INTERFACE PUBLIC MoveVelocityBuilder EXTENDS __System.IQueryInterface

METHOD PUBLIC Acceleration : MoveVelocityBuilder
VAR_INPUT
	value : LREAL;
END_VAR
END_METHOD

METHOD PUBLIC BufferMode : MoveVelocityBuilder
VAR_INPUT
	mode : MotionBufferMode;
END_VAR
END_METHOD

METHOD PUBLIC BuildMoveVelocityCommand : MotionCommand
VAR_INPUT
	axis : Axis;
END_VAR
END_METHOD

METHOD PUBLIC Deceleration : MoveVelocityBuilder
VAR_INPUT
	value : LREAL;
END_VAR
END_METHOD

METHOD PUBLIC Distance : MoveRelativeBuilder
VAR_INPUT
	value : LREAL;
END_VAR
END_METHOD

METHOD PUBLIC Jerk : MoveVelocityBuilder
VAR_INPUT
	value : LREAL;
END_VAR
END_METHOD

METHOD PUBLIC Position : MoveAbsoluteBuilder
VAR_INPUT
	value : LREAL;
END_VAR
END_METHOD

METHOD PUBLIC Velocity : MoveVelocityBuilder
VAR_INPUT
	value : LREAL;
END_VAR
END_METHOD

END_INTERFACE

(* stored: Version 1.1.0.1
   Itf MoveVelocityBuilder: Id {af81a36f-91e0-4229-8050-674aaf4d51c8}
   Folder Builders: Id {7fd778aa-403b-4bcf-b94b-ddb110cd0772}
   Folder PropertySetters: Id {c78165b8-d771-464a-881b-28b518193161}
   Method Acceleration: Id {1a50edb1-113b-4f46-83c6-b8f26a71a15e}
   Method BufferMode: Id {6a4f0400-b046-43df-b9ee-74e7ee22d50a}
   Method BuildMoveVelocityCommand: Id {0fd3c392-d1e2-06f3-2fa5-d8869d117ef5}
   Method Deceleration: Id {2885aa42-90e4-4613-82d7-1c22ebf0dd39}
   Method Distance: Id {492191b7-499f-40fe-a63e-283905023ebf}
   Method Jerk: Id {d31e94a9-727f-4bfb-bd51-0dd8ad61940f}
   Method Position: Id {2aad1022-9d1b-4af0-bc07-544790ecfdea}
   Method Velocity: Id {eb1b270e-f436-450a-b153-6c07dbc75ac9} *)
